// TIA Portal V18 export
DATA_BLOCK "Pump & Flowrate"   // DB48
{ S7_Optimized_Access := 'TRUE' }
VERSION : 0.1
// stored: AutoNumber true, DBAccessibleFromOPCUA true, IsOnlyStoredInLoadMemory false, IsRetainMemResEnabled false, IsWriteProtectedInAS false, MemoryReserve 100
   VAR RETAIN
      "Pump A" : Struct
         size : Real := 0.0590186;
         "Pump Speed" : Int := 200;
         "speed sensor impulse" : Int := 0;
         "size in ml" : Real := 0.0590186;
         "serial number" : String[20] := '';
      END_STRUCT;
      "Pump B" : Struct
         size : Real := 0.0546615;
         "size in ml" : Real := 0.0546615;
         "Pump Speed" : Int := 200;
         "speed sensor impulse" : Int := 0;
         "serial number" : String[20] := '';
      END_STRUCT;
   END_VAR
   VAR
      capacity : Struct
         "Pump A" : Real := 11.80372;
         "pump B in ml" : Real := 10.9323;
         "pump A in ml" : Real := 11.80372;
         "pump B" : Real := 10.9323;
      END_STRUCT;
      "Flowrate Input" : Struct
         "Pump A" : Real := 5.0;
         "Pump A in ml" : Real := 5.0;
         "pump B in ml" : Real := 2.0;
         "Pump B" : Real := 2.0;
      END_STRUCT;
      "mixed flowrate Input" : Real := 6.0;
      "Qty input" : Real := 0.5;
      "Calculated flowrate A with adjustment" : Real := 4.0;
      "Calculated Flowrate B  with adjustment" : Real := 2.0;
      "Calculated flowrate A without adjustment" : Real := 4.0;
      "Calculated Flowrate B without adjustment" : Real := 2.0;
      "Flowrate Adjustment A" : Real := 0.0;
      "Flowrate Adjustment B" : Real := 0.0;
      "Metering time calculated" : DInt := 5000;
      "Mixed Flowrate maximum" : Real := 0.0;
      "metering time in seconds" : Int := 5;
      "fowrate A Adjustment Configuration" : Real := 0.0;
      "fowrate B Adjustment Configuration" : Real := 0.0;
      "Maximum Mixed Flowrate" : Real := 17.70558;
      "Minimum Mixed Flowrate" : Real := 0.1062335;
      "Pump A minimum Flowrate" : Real := 1.180372;
      "Pump B minimum Flowrate" : Real := 1.09323;
      "Flush Maximum Flowrate" : Real := 10.9323;
      "Flush minimum Flowrate" : Real := 1.09323;
      startSnuff_Back_PumpA : Bool := TRUE;
      startSnuff_Back_PumpB : Bool := TRUE;
      SnuffBack_SpeedA : Bool := FALSE;
   END_VAR
   VAR RETAIN
      referenceRamp_PumpA : Real := 6000.0;
      referenceRamp_PumpB : Real := 6000.0;
      PumpsizeA_original : Real := 0.05;
      PumpsizeB_original : Real := 0.05;
   END_VAR
   VAR
      pumpA_edited : Bool := FALSE;
      pumpB_edited : Bool := FALSE;
      record_size : Bool := FALSE;
   END_VAR
BEGIN
END_DATA_BLOCK
